// TIA Portal V18 export
FUNCTION_BLOCK "cycle_point_to_point"   // FB51, FBD
{ S7_Optimized_Access := 'TRUE' }
VERSION : 0.1
// stored: AutoNumber true, IsIECCheckEnabled false, IsRetainMemResEnabled false, MemoryReserve 100, SetENOAutomatically false, UDAEnableTagReadback false
   VAR
      saved_points : Bool;
      defect_points : Bool;
   END_VAR
BEGIN
END_FUNCTION_BLOCK
